TYPE EtcMasterBase_62654B43 :
STRUCT
END_STRUCT
END_TYPE

(* stored: Version 1.2.0.0, ProductVersion 3.1.4024.11
   DUT EtcMasterBase_62654B43: Id {f655ce51-b2bc-42f0-a9fb-361a11843ddc} *)
